Omron Sysmac Studio project Test3 (Sysmac Studio 1.56.0.64011, StandardProject)

# Controller new_Controller_0: NX1P2-1040DT1 version 1.16
Task PrimaryTask (priority 4, period or condition 2000): Program0

VAR_GLOBAL
    BIO_Input_Bit_00 : BOOL;  (* at BuiltInIO://cpu/#0/Input_Bit_00 *)
    BIO_Input_Bit_01 : BOOL;  (* at BuiltInIO://cpu/#0/Input_Bit_01 *)
    BIO_Input_Bit_02 : BOOL;  (* at BuiltInIO://cpu/#0/Input_Bit_02 *)
    Start : BOOL;
    Stop : BOOL;
    Çıkış : BOOL;
    Motor : BOOL;
    Start2 : BOOL;
    Motorİleri : BOOL;
    Motor_İleri : BOOL;
    Motor_Geri : BOOL;
END_VAR

PROGRAM Program0
VAR
    Motor_Temp1 : BOOL;
    Motor_Temp2 : BOOL;
END_VAR
VAR_EXTERNAL
    Start : BOOL;
    Stop : BOOL;
    Çıkış : BOOL;
    Motor : BOOL;
    BIO_Input_Bit_00 : BOOL;
    BIO_Input_Bit_01 : BOOL;
    BIO_Input_Bit_02 : BOOL;
    Start2 : BOOL;
    Motorİleri : BOOL;
    Motor_İleri : BOOL;
    Motor_Geri : BOOL;
END_VAR

(* Section InOut: ladder, written here as Structured Text *)

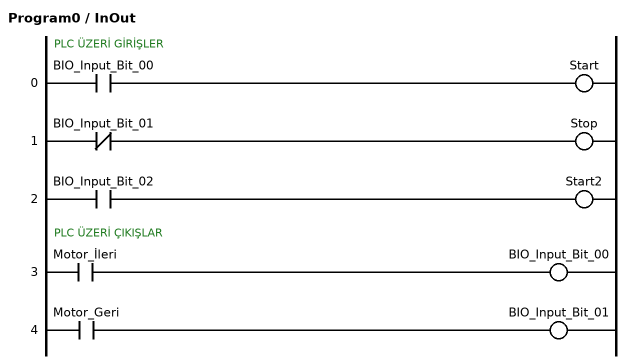
(* Rung 0: PLC ÜZERİ GİRİŞLER *)
Start := BIO_Input_Bit_00;
(* Rung 1 *)
Stop := NOT BIO_Input_Bit_01;
(* Rung 2 *)
Start2 := BIO_Input_Bit_02;
(* Rung 3: PLC ÜZERİ ÇIKIŞLAR *)
BIO_Input_Bit_00 := Motor_İleri;
(* Rung 4 *)
BIO_Input_Bit_01 := Motor_Geri;

(* Section Section1: ladder, written here as Structured Text *)

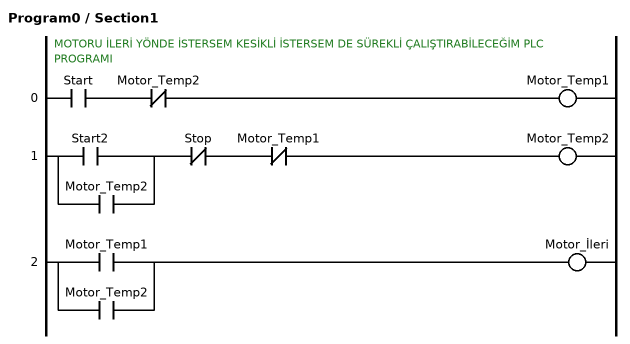
(* Rung 0: MOTORU İLERİ YÖNDE İSTERSEM KESİKLİ İSTERSEM DE SÜREKLİ ÇALIŞTIRABİLECEĞİM PLC PROGRAMI *)
Motor_Temp1 := Start AND NOT Motor_Temp2;
(* Rung 1 *)
Motor_Temp2 := (Start2 OR Motor_Temp2) AND NOT Stop AND NOT Motor_Temp1;
(* Rung 2 *)
Motor_İleri := Motor_Temp1 OR Motor_Temp2;
END_PROGRAM